FUNCTION_BLOCK FB_ResetAll
VAR_INPUT
	bExecute : BOOL;
END_VAR
VAR_OUTPUT
	bDone : BOOL;
	bError : BOOL;
END_VAR
VAR
	reset1 : MC_Reset;
	reset2 : MC_Reset;
END_VAR
VAR_IN_OUT
	io_M1 : AXIS_REF;
	io_M2 : AXIS_REF;
END_VAR

reset1(Axis := io_M1, Execute := bExecute);
reset2(Axis := io_M2, Execute := bExecute);

bError := reset1.Error OR reset2.Error;
bDone := reset1.Done AND reset2.Done AND NOT bError;

END_FUNCTION_BLOCK

(* stored: Version 1.1.0.1, ProductVersion 3.1.4024.9
   POU FB_ResetAll: Id {553be986-174c-4702-a8c0-5d361719b831}, SpecialFunc None *)
